(* CODESYS project fbMotorV1.project

Project tree, tasks and I/O mapping:
  Device : CODESYS Control Win V3, 3S - Smart Software Solutions GmbH, version 3.5.17.0
    application Application
      libraries: VisuDialogs, * (System)
      task VISU_TASK (cyclic, interval 100 ms, priority 10) calls VisuElems.Visu_Prg
      task Task (cyclic, interval t#4ms, priority 1) calls manipulateST
      program MOTION_PRG [FBD]
      Cam1
      visualisation Visualization
      Cam2
      program Cammanipulation [FBD]
      program Evedon [FBD]
      program Konumagit [FBD]
      Cam3
      program manipulateST [ST]
      program POWER [ST]
    SoftMotion General Axis Pool : SoftMotion General Axis Pool, 3S - Smart Software Solutions GmbH, version 4.11.0.0
      Drive : SM_Drive_Virtual, 3S - Smart Software Solutions GmbH, order no. 1805, version 4.0.0.0
          settings: wDriveID = 0; iMovementType = 0; fSWMaxVelocity = 1e3; fSWMaxAcceleration = 1e5; fSWMaxDeceleration = 1e5; fRampJerk = 1e7; fSWLimitPositive = 100.0
      Virtual : SM_Drive_Virtual, 3S - Smart Software Solutions GmbH, order no. 1805, version 4.0.0.0
          settings: iMovementType = 0; fPositionPeriod = 360; fSWMaxVelocity = 1e3; fSWMaxAcceleration = 1e5; fSWMaxDeceleration = 1e5; fRampJerk = 1e7
      Drayv : SM_Drive_Virtual, 3S - Smart Software Solutions GmbH, order no. 1805, version 4.0.0.0
          settings: wDriveID = 2; iMovementType = 0; fSWMaxVelocity = 1e3; fSWMaxAcceleration = 1e5; fSWMaxDeceleration = 1e5
  libraries: Standard, 3.5.18.0 (System)
  text list GlobalTextList
  GlobalImagePool
*)

// Device/Application/manipulateST
PROGRAM manipulateST
VAR
//SERVO ON
power1,power2 : MC_POWER;
Cam3: ARRAY[0..3] OF SMC_CAMXYVA := [
        (dX := 0, dY := 0, dV := 0, dA := 0),
        (dX := 120, dY := 120, dV := 1, dA := 0),
        (dX := 240, dY := 350, dV := 2, dA := 0),
        (dX := 360, dY := 360, dV := 0, dA := 0)];
		//Ust kisimdaki degerler yerine degisken atayarak
		//cam tablosunu makine calisir iken guncelleyebiliriz.
	Cam: MC_CAM_REF := (nElements := 4, byType := 3, xStart := 0, 
	xEnd := 360, nTappets := 0, strCAMName := 'Cam3', 
	pce := ADR(Cam3), xPartofLM := TRUE);
	CamSet: SMC_GetCamSlaveSetPosition;
	MoveVirtual: MC_MoveVelocity;
	TableSelect: MC_CamTableSelect; 
	CamIn: MC_CamIn; 
	
	
	EXE: BOOL;
	SETLE:BOOL;
	MasterSpeed : LREAL;
	MasterAcc : LREAL;
	MasterDec: LREAL;

END_VAR

//SERVO POWER BLOCKS
power1(Axis := Virtual);
power1.Enable:= TRUE;
power1.bRegulatorOn:=TRUE;
power1.bDriveStart:= TRUE;
power2(Axis:=Drive);
power2.Enable:= TRUE;
power2.bRegulatorOn:=TRUE;
power2.bDriveStart:= TRUE;

//FOR MASTER AXIS VIRTUAL MOVEMENT
MoveVirtual(Axis := Virtual);

MoveVirtual.Execute := EXE AND power2.Status;
MoveVirtual.Velocity := MasterSpeed;
MoveVirtual.Acceleration := MasterAcc;
MoveVirtual.Deceleration := MasterDec;
MoveVirtual.Direction := Positive;

//FOR SELECTING CUSTOM CAM TABLE
TableSelect(Master:= Virtual, Slave:= Drive,CamTable:= Cam);

TableSelect.Execute := TRUE;
TableSelect.Periodic := TRUE;
TableSelect.MasterAbsolute := TRUE;
TableSelect.SlaveAbsolute := TRUE;

//FOR USING CAM TABLE
CamIn(Master := Virtual, Slave := Drive);

CamIn.Execute := power1.Status;
CamIn.MasterOffset := 0;
CamIn.SlaveOffset := 0;
CamIn.MasterScaling := 1;
CamIn.SlaveScaling := 1;
CamIn.StartMode := absolute;
CamIn.CamTableID := TableSelect.CamTableID;
CamIn.VelocityDiff := 1;
CamIn.Acceleration := 1;
CamIn.Deceleration := 1;
CamIn.TappetHysteresis := 1;

CamSet(Master:= Virtual, Slave := Drive);
CamSet.Enable := SETLE;
CamSet.MasterOffset:= 10;
CamSet.SlaveOffset:= 10;
CamSet.MasterScaling:= 10;
CamSet.SlaveScaling:= 10;
CamSet.CamTableID:= TableSelect.CamTableID;

END_PROGRAM

// Device/Application/POWER
PROGRAM POWER
VAR
	//servolarin ON konumuna gelmesi icin mutlaka calismali.
	power1,power2,power3 : MC_POWER;
END_VAR

power1.Enable:= TRUE;
power1.Axis := Drive;
power1.bRegulatorOn:=TRUE;
power1.bDriveStart:= TRUE;

power2.Enable:= TRUE;
power2.Axis := Drive;
power2.bRegulatorOn:=TRUE;
power2.bDriveStart:= TRUE;

power3.Enable:= TRUE;
power3.Axis := Drive;
power3.bRegulatorOn:=TRUE;
power3.bDriveStart:= TRUE;

END_PROGRAM

// Device/Application/MOTION_PRG
PROGRAM MOTION_PRG
VAR
	power1, power2, power3: MC_Power; //servolarin ON konumuna gelmesi icin mutlaka calismali.
	TableSelect,TableSelect2: MC_CamTableSelect; //istenen cam tablosunu secmeye yarar.
	CamIn,CamIn2: MC_CamIn; //secildikten sonra cam tablosunu devreye alir.
	Tappet,Tappet2: SMC_GetTappetValue;
	MoveVirtual: MC_MoveVelocity; //Istenen hizda doner, stop gelmedigi surece ayni hizda devam eder.
	FA: BOOL;
	M1: BOOL; //baslatmak icin setle durdurmak icin resetle
END_VAR

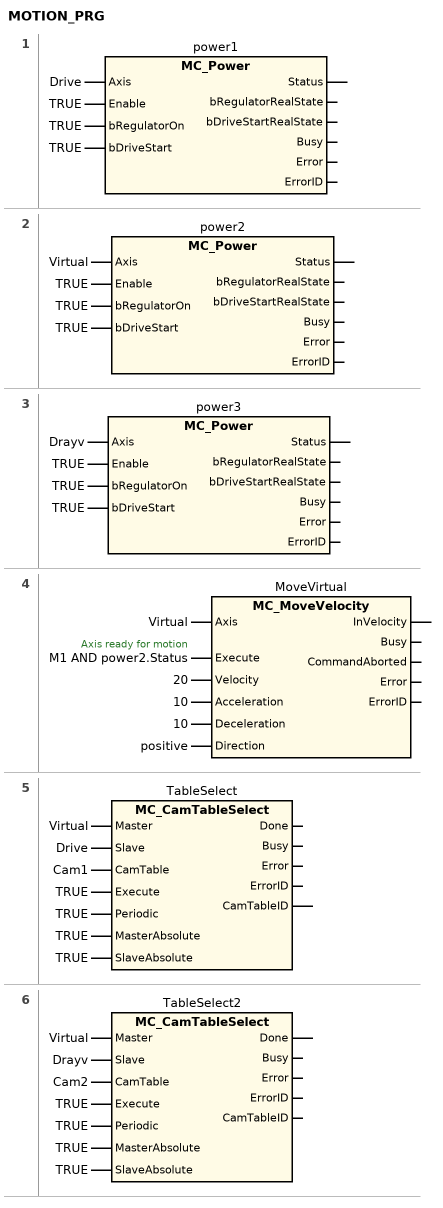
// NETWORK 1
power1(Axis := Drive, Enable := TRUE, bRegulatorOn := TRUE, bDriveStart := TRUE); // MC_Power

// NETWORK 2
power2(Axis := Virtual, Enable := TRUE, bRegulatorOn := TRUE, bDriveStart := TRUE); // MC_Power

// NETWORK 3
power3(Axis := Drayv, Enable := TRUE, bRegulatorOn := TRUE, bDriveStart := TRUE); // MC_Power

// NETWORK 4
//   M1 AND power2.Status: Axis ready for motion
MoveVirtual(
    Axis := Virtual,
    Execute := M1 AND power2.Status,
    Velocity := 20,
    Acceleration := 10,
    Deceleration := 10,
    Direction := positive); // MC_MoveVelocity

// NETWORK 5
TableSelect(
    Master := Virtual,
    Slave := Drive,
    CamTable := Cam1,
    Execute := TRUE,
    Periodic := TRUE,
    MasterAbsolute := TRUE,
    SlaveAbsolute := TRUE); // MC_CamTableSelect

// NETWORK 6
TableSelect2(
    Master := Virtual,
    Slave := Drayv,
    CamTable := Cam2,
    Execute := TRUE,
    Periodic := TRUE,
    MasterAbsolute := TRUE,
    SlaveAbsolute := TRUE); // MC_CamTableSelect

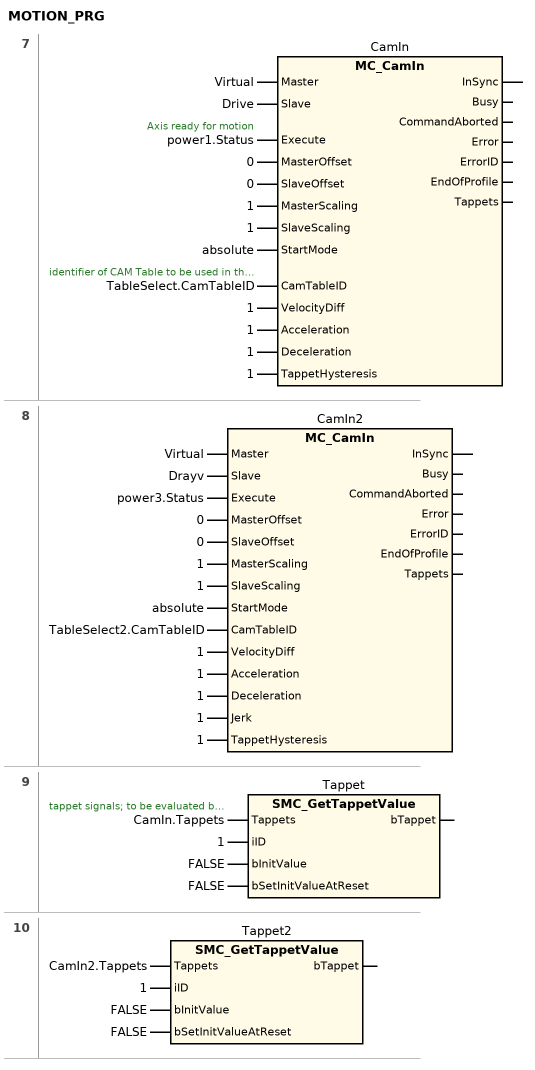
// NETWORK 7
//   power1.Status: Axis ready for motion
//   TableSelect.CamTableID: identifier of CAM Table to be used in the MC_CamIn FB
CamIn(
    Master := Virtual,
    Slave := Drive,
    Execute := power1.Status,
    MasterOffset := 0,
    SlaveOffset := 0,
    MasterScaling := 1,
    SlaveScaling := 1,
    StartMode := absolute,
    CamTableID := TableSelect.CamTableID,
    VelocityDiff := 1,
    Acceleration := 1,
    Deceleration := 1,
    TappetHysteresis := 1); // MC_CamIn

// NETWORK 8
CamIn2(
    Master := Virtual,
    Slave := Drayv,
    Execute := power3.Status,
    MasterOffset := 0,
    SlaveOffset := 0,
    MasterScaling := 1,
    SlaveScaling := 1,
    StartMode := absolute,
    CamTableID := TableSelect2.CamTableID,
    VelocityDiff := 1,
    Acceleration := 1,
    Deceleration := 1,
    Jerk := 1,
    TappetHysteresis := 1); // MC_CamIn

// NETWORK 9
//   CamIn.Tappets: tappet signals; to be evaluated by MC_GetTappetValue FBs
Tappet(Tappets := CamIn.Tappets, iID := 1, bInitValue := FALSE, bSetInitValueAtReset := FALSE); // SMC_GetTappetValue

// NETWORK 10
Tappet2(Tappets := CamIn2.Tappets, iID := 1, bInitValue := FALSE, bSetInitValueAtReset := FALSE); // SMC_GetTappetValue

END_PROGRAM

// Device/Application/Cammanipulation
PROGRAM Cammanipulation
VAR
	Cam3: ARRAY[0..3] OF SMC_CAMXYVA := [
        (dX := 0, dY := 0, dV := 0, dA := 0),
        (dX := 120, dY := 120, dV := 1, dA := 0),
        (dX := 240, dY := 350, dV := 2, dA := 0),
        (dX := 360, dY := 360, dV := 0, dA := 0)];
		//Ust kisimdaki degerler yerine degisken atayarak
		//cam tablosunu makine calisir iken guncelleyebiliriz.
	Cam: MC_CAM_REF := (nElements := 4, byType := 3, xStart := 0, 
	xEnd := 360, nTappets := 0, strCAMName := 'Cam3', 
	pce := ADR(Cam3), xPartofLM := TRUE);
	power1, power2 : MC_Power; 
	//SMC_GetCamSlaveSetPosition_0: SMC_GetCamSlaveSetPosition;
	MoveVirtual: MC_MoveVelocity;
	TableSelect: MC_CamTableSelect; 
	CamIn: MC_CamIn; 
	SETLE: BOOL;
	EXE: BOOL;
	CamSet: SMC_GetCamSlaveSetPosition;
END_VAR

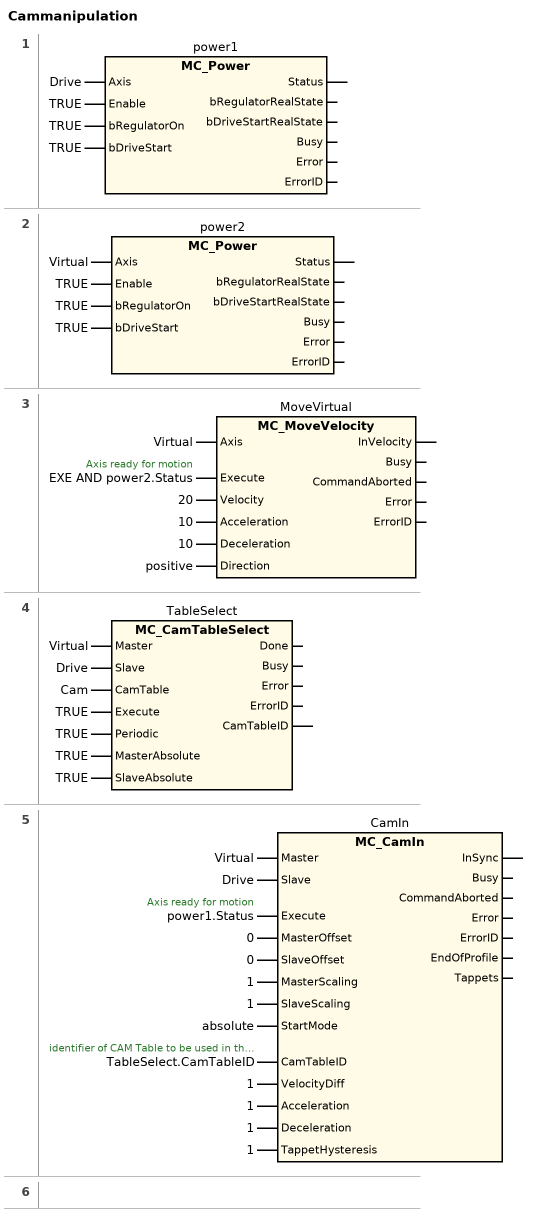
// NETWORK 1
power1(Axis := Drive, Enable := TRUE, bRegulatorOn := TRUE, bDriveStart := TRUE); // MC_Power

// NETWORK 2
power2(Axis := Virtual, Enable := TRUE, bRegulatorOn := TRUE, bDriveStart := TRUE); // MC_Power

// NETWORK 3
//   EXE AND power2.Status: Axis ready for motion
MoveVirtual(
    Axis := Virtual,
    Execute := EXE AND power2.Status,
    Velocity := 20,
    Acceleration := 10,
    Deceleration := 10,
    Direction := positive); // MC_MoveVelocity

// NETWORK 4
TableSelect(
    Master := Virtual,
    Slave := Drive,
    CamTable := Cam,
    Execute := TRUE,
    Periodic := TRUE,
    MasterAbsolute := TRUE,
    SlaveAbsolute := TRUE); // MC_CamTableSelect

// NETWORK 5
//   power1.Status: Axis ready for motion
//   TableSelect.CamTableID: identifier of CAM Table to be used in the MC_CamIn FB
CamIn(
    Master := Virtual,
    Slave := Drive,
    Execute := power1.Status,
    MasterOffset := 0,
    SlaveOffset := 0,
    MasterScaling := 1,
    SlaveScaling := 1,
    StartMode := absolute,
    CamTableID := TableSelect.CamTableID,
    VelocityDiff := 1,
    Acceleration := 1,
    Deceleration := 1,
    TappetHysteresis := 1); // MC_CamIn

// NETWORK 6

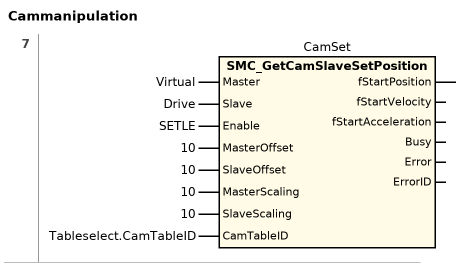
// NETWORK 7
CamSet(
    Master := Virtual,
    Slave := Drive,
    Enable := SETLE,
    MasterOffset := 10,
    SlaveOffset := 10,
    MasterScaling := 10,
    SlaveScaling := 10,
    CamTableID := Tableselect.CamTableID); // SMC_GetCamSlaveSetPosition

END_PROGRAM

// Device/Application/Evedon
PROGRAM Evedon
VAR
	M4: BOOL;
	SMC_Homing_0: SMC_Homing; // referans sensor/aygit TRUE sinyali verene kadar doner, sinyal gelince
	//o konumu HOME olarak kabul eder ve poizsyon kismina ne girildi ise orayi o pozisyon kabul eder.
	Drayv_Home_Yavas: LREAL;
	Drayv_Home_Hizli: LREAL;
	Drayv_Home_Sensor: BOOL;
	MC_Home_0: MC_Home;
	M8: BOOL;
	JOGDrayv: MC_Jog;
	FORW: BOOL;
	REVE: BOOL;
END_VAR

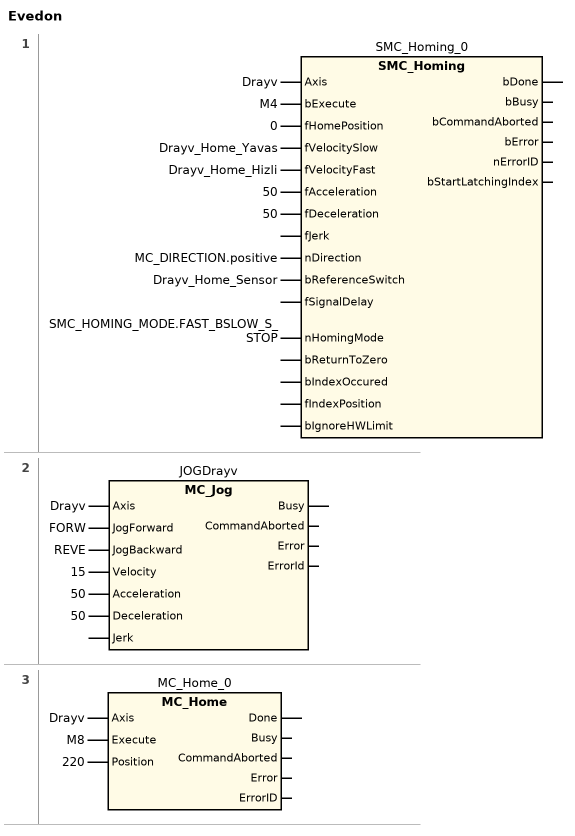
// NETWORK 1
SMC_Homing_0(
    Axis := Drayv,
    bExecute := M4,
    fHomePosition := 0,
    fVelocitySlow := Drayv_Home_Yavas,
    fVelocityFast := Drayv_Home_Hizli,
    fAcceleration := 50,
    fDeceleration := 50,
    nDirection := MC_DIRECTION.positive,
    bReferenceSwitch := Drayv_Home_Sensor,
    nHomingMode := SMC_HOMING_MODE.FAST_BSLOW_S_STOP); // SMC_Homing

// NETWORK 2
JOGDrayv(
    Axis := Drayv,
    JogForward := FORW,
    JogBackward := REVE,
    Velocity := 15,
    Acceleration := 50,
    Deceleration := 50); // MC_Jog

// NETWORK 3
MC_Home_0(Axis := Drayv, Execute := M8, Position := 220); // MC_Home

END_PROGRAM

// Device/Application/Konumagit
PROGRAM Konumagit
VAR
	MC_MoveRelative_0: MC_MoveRelative; //motoru istenen miktarda dondurur sonra durur. 
	//tekrar tetiklenecek olursa, kaldigi yerden baslar yine istenen miktarda dondurur.
	relativ: BOOL;
	Veloc: LREAL;
	distan: LREAL;
END_VAR

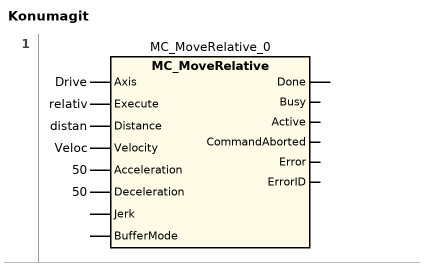
// NETWORK 1
MC_MoveRelative_0(
    Axis := Drive,
    Execute := relativ,
    Distance := distan,
    Velocity := Veloc,
    Acceleration := 50,
    Deceleration := 50); // MC_MoveRelative

END_PROGRAM

// Device/Application/Visualization
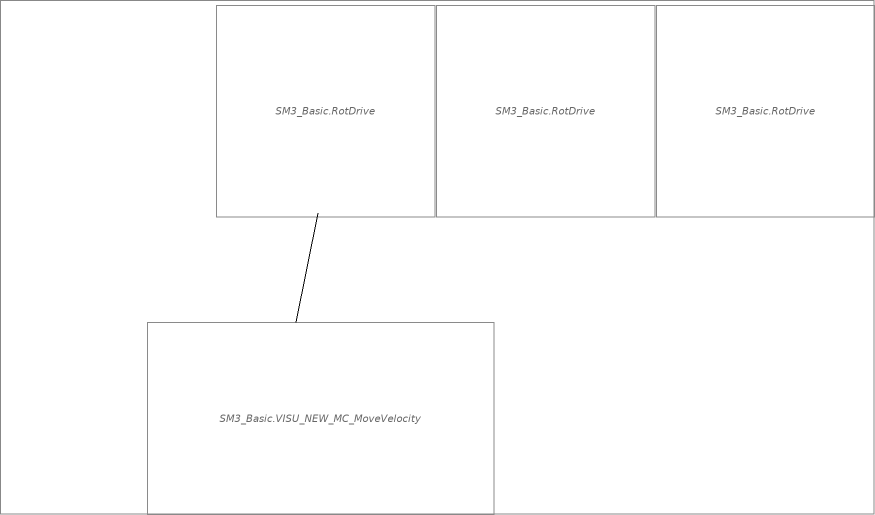
VISUALIZATION Visualization  // 875x515
    Frame (147,322 347x193)
        shows SM3_Basic.VISU_NEW_MC_MoveVelocity(m_Input_FB := MOTION_PRG.MoveVirtual)
    Frame (216,5 219x212)
        shows SM3_Basic.RotDrive(m_Input_AXISREF := Virtual)
    Frame (436,5 219x212)
        shows SM3_Basic.RotDrive(m_Input_AXISREF := Drive)
    Frame (656,5 219x212)
        shows SM3_Basic.RotDrive(m_Input_AXISREF := Drayv)
    Line (84,136)
    Line (296,322) (318,213)
END_VISUALIZATION
